(* CODESYS project addition_2.xml

Project tree, tasks and I/O mapping:
  function addition_2 [ST]
*)

// addition_2
FUNCTION addition_2 : Bool
VAR_INPUT
	KEKEKE:BOOL;
END_VAR
VAR
	tempVar64:STRING;
END_VAR

addition_2 := FALSE;
tempVar64	:=	'YOYOYOY';
addition_2		:=		KEKEKE;

END_FUNCTION
